VAR_GLOBAL
	//Better have your inputs and outputs!
	// M1L0
	Serial_stComIn_M1L0   AT %I*	:	EL6inData22B (*KL6inData22B*);
	Serial_stComOut_M1L0  AT %Q*	:	EL6outData22B (*KL6outData22B*);

	// M2L0
	Serial_stComIn_M2L0   AT %I*	:	EL6inData22B (*KL6inData22B*);
	Serial_stComOut_M2L0  AT %Q*	:	EL6outData22B (*KL6outData22B*);
END_VAR

(* stored: Version 1.1.0.1, ProductVersion 3.1.4022.18
   GVL GVL_SerialIO: Id {e2338c89-1965-407c-b604-590f80e0dc24} *)
